(* IEC 61131-3 sources: CodigoPPC/FB Auxiliares, 7 files *)

(* ---- FB_CheckInversores.st ---- *)
// ════════════════════════════════════════════════════════════════════
// FB_CheckInversores — Varredura de presença de inversores no startup
// ════════════════════════════════════════════════════════════════════
//
// Responsabilidade:
//   Percorrer sequencialmente todos os inversores configurados
//   (InvActivePower > 0) em COM1 e COM2, disparar 1 transação
//   Modbus em cada um e verificar ACK. Não valida o valor lido.
//
// Critério de avanço:
//   respondidos / configurados >= GVL_Persis.InvCheckThreshold → xDone=TRUE
//   abaixo do limiar ou timeout global                         → xFailed=TRUE
//
// Contrato com FB_Startup:
//   • xEnable := TRUE  para iniciar/continuar a varredura
//   • xEnable := FALSE reseta o FB (pronto para nova execução)
//   • Lê resultado via xDone / xFailed a cada ciclo
//   • xFailed=TRUE: ler uRespondedTotal e uConfiguredTotal para log
//
// Restrições:
//   • 1 transação Modbus por ciclo de scan (sequencial, determinístico)
//   • Não escreve em GVL_ALARM_MANAGER — responsabilidade do FB_Startup
//   • Tempo máximo: TimeInvTimeout (default 60s para até 30 inversores)
// ════════════════════════════════════════════════════════════════════
FUNCTION_BLOCK FB_CheckInversores

VAR_INPUT
    xEnable         : BOOL;             // TRUE = executar; FALSE = reset
    tTxTimeout      : TIME := T#500MS;  // timeout por transação individual
    tGlobalTimeout  : TIME := T#60S;    // timeout para varredura completa
END_VAR

VAR_OUTPUT
    xDone           : BOOL;             // varredura concluída e acima do limiar
    xFailed         : BOOL;             // abaixo do limiar ou timeout global
    uRespondedTotal : UINT;             // total de inversores que responderam
    uConfiguredTotal: UINT;             // total de inversores configurados
    uLastFailIdx    : UINT;             // índice do último inversor que não respondeu
    uLastFailCOM    : UINT;             // canal do último inversor que não respondeu (1 ou 2)
END_VAR

VAR
    fbTx            : FB_ModBus;        // instância única reutilizada ciclo a ciclo
    uCheckIdx       : UINT := 1;        // índice atual (1..15 dentro do canal)
    uCheckCOM       : UINT := 1;        // canal atual: 1=COM1, 2=COM2, 3=avaliação final
    uRespondedCOM1  : UINT := 0;
    uRespondedCOM2  : UINT := 0;
    bInitDone       : BOOL := FALSE;    // guarda de inicialização
    TonGlobal       : TON;
    // ── Startup: verificação de presença de inversores ────────────
    // Fração mínima de inversores que devem responder para avançar o startup.
    // 1.0 = todos devem responder (padrão conservador)
    // 0.8 = pelo menos 80% devem responder
    CheckThreshold  : REAL := 1.0;
END_VAR

    // ── Reset quando desabilitado ─────────────────────────────────────
    IF NOT xEnable THEN
        xDone            := FALSE;
        xFailed          := FALSE;
        uRespondedCOM1   := 0;
        uRespondedCOM2   := 0;
        uRespondedTotal  := 0;
        uConfiguredTotal := 0;
        uLastFailIdx     := 0;
        uLastFailCOM     := 0;
        uCheckIdx        := 1;
        uCheckCOM        := 1;
        bInitDone        := FALSE;
        TonGlobal(IN := FALSE);
        RETURN;
    END_IF

    // ── Se já terminou, mantém resultado sem re-executar ─────────────
    IF xDone OR xFailed THEN
        RETURN;
    END_IF

    // ── Inicialização na primeira entrada ────────────────────────────
    IF NOT bInitDone THEN
        uConfiguredTotal := GVL_Main.NInversoresCOM01 + GVL_Main.NInversoresCOM02;
        bInitDone        := TRUE;

        // COM2 vazio é permitido — varredura só em COM1
        // uCheckCOM já = 1, sem ação adicional
    END_IF

    // ── Timeout global ────────────────────────────────────────────────
    TonGlobal(IN := TRUE, PT := tGlobalTimeout);
    IF TonGlobal.Q THEN
        TonGlobal(IN := FALSE);
        uRespondedTotal := uRespondedCOM1 + uRespondedCOM2;
        xFailed := TRUE;
        RETURN;
    END_IF

    // ── Varredura COM1 ────────────────────────────────────────────────
    IF uCheckCOM = 1 THEN

        IF uCheckIdx <= GVL_Main.NInversoresCOM01 THEN
            fbTx(
                tTimeout := tTxTimeout,
                trigInv  := GVL_Main.trigInvCOM100[uCheckIdx, 0],
                pSlave   := GVL_Main.pInversores100[uCheckIdx]^
            );

            CASE fbTx.result OF
                E_ModbusResult.DONE:
                    uRespondedCOM1 := uRespondedCOM1 + 1;
                    uCheckIdx      := uCheckIdx + 1;

                E_ModbusResult.ERRO,
                E_ModbusResult.TIMEOUT:
                    uLastFailIdx := uCheckIdx;
                    uLastFailCOM := 1;
                    uCheckIdx    := uCheckIdx + 1;

                // BUSY: aguarda sem avançar
            END_CASE

        ELSE
            // COM1 concluída
            uCheckIdx := 1;
            uCheckCOM := 2;  // avança para COM2 (mesmo que vazia — avaliação em uCheckCOM=3)
        END_IF

    // ── Varredura COM2 ────────────────────────────────────────────────
    ELSIF uCheckCOM = 2 THEN

        IF GVL_Main.NInversoresCOM02 = 0 THEN
            // Canal vazio — pula direto para avaliação
            uCheckCOM := 3;

        ELSIF uCheckIdx <= GVL_Main.NInversoresCOM02 THEN
            fbTx(
                tTimeout := tTxTimeout,
                trigInv  := GVL_Main.trigInvCOM200[uCheckIdx, 0],
                pSlave   := GVL_Main.pInversores200[uCheckIdx]^
            );

            CASE fbTx.result OF
                E_ModbusResult.DONE:
                    uRespondedCOM2 := uRespondedCOM2 + 1;
                    uCheckIdx      := uCheckIdx + 1;

                E_ModbusResult.ERRO,
                E_ModbusResult.TIMEOUT:
                    uLastFailIdx := uCheckIdx;
                    uLastFailCOM := 2;
                    uCheckIdx    := uCheckIdx + 1;

                // BUSY: aguarda sem avançar
            END_CASE

        ELSE
            // COM2 concluída
            uCheckCOM := 3;
        END_IF

    // ── Avaliação final ───────────────────────────────────────────────
    ELSIF uCheckCOM = 3 THEN

        TonGlobal(IN := FALSE);
        uRespondedTotal := uRespondedCOM1 + uRespondedCOM2;

        IF uConfiguredTotal = 0 THEN
            // Proteção defensiva — não deveria chegar aqui (stInit já bloqueia)
            xFailed := TRUE;
            RETURN;
        END_IF

        IF (TO_REAL(uRespondedTotal) / TO_REAL(uConfiguredTotal)) >= CheckThreshold THEN
            xDone := TRUE;
        ELSE
            xFailed := TRUE;
        END_IF

    END_IF

END_FUNCTION_BLOCK

(* ---- FB_ModBus.st ---- *)
FUNCTION_BLOCK FB_ModBus

VAR_INPUT
    tTimeout    : TIME;
END_VAR

VAR_IN_OUT
    trigInv     : BOOL;                    // ex.: Global.trigInvCOM100[i]
    pSlave      : ModbusSlaveComPort;      // ex.: Global.pInversores100[i]^
END_VAR

VAR_OUTPUT
    result      : E_ModbusResult;
END_VAR

VAR
    state       : (TRIG, WAIT_BUSY_ON, WAIT_DONE) := TRIG;
    tonTimer    : TON;
END_VAR

    // ============================================================
    // Máquina de estados de escrita em inversores
    // ============================================================

    // estado default por ciclo
    result := E_ModbusResult.BUSY;

    // timeout só enquanto espera finalização real
    tonTimer(IN := (state = WAIT_DONE), PT := tTimeout);

    CASE state OF

        TRIG:
            trigInv := TRUE;
            state := WAIT_BUSY_ON;

       WAIT_BUSY_ON:
            trigInv := FALSE;            // desce trigger (garante borda)
            IF pSlave.xBusy THEN         // transação realmente iniciou
                state := WAIT_DONE;
            END_IF

        WAIT_DONE:
        	IF pSlave.xDone THEN
                trigInv := FALSE;
                state := TRIG;
                result := E_ModbusResult.DONE;

          	ELSIF pSlave.xError THEN
                state := TRIG;
    			trigInv := FALSE;
                result := E_ModbusResult.ERRO;
    			FC_LogEvent(
    				eCode:=TO_UINT(pSlave.byModbusError) + 16#4A00,
    				bRaised:=TRUE,
    				rParam1:=0.0,
    				rParam2:=0.0,
    				uMachState := GVL_Main.MachineState
    				);

          	ELSIF tonTimer.Q THEN
                state := TRIG;
                trigInv := FALSE;
                result := E_ModbusResult.TIMEOUT;
            END_IF
    END_CASE
END_FUNCTION_BLOCK

(* ---- FB_SetRTC.st ---- *)
(*
================================================================================
  FB_SetRTC — Correção de Data/Hora do RTC via IHM
================================================================================
  Propósito:
    Permite que o operador corrija o relógio do CLP (WAGO CC100) diretamente
    pela IHM, sem necessidade de acesso ao Codesys IDE.

  Problema resolvido:
    O CC100 não possui bateria de RTC confiável. Após queda de energia, o
    relógio retorna para 1970-01-01 00:00:00. Isso corrompe o agendamento
    (FB_Scheduler), o log de eventos e qualquer registro com timestamp.

  Comportamento:
    1. O operador preenche os campos de data/hora na IHM e aciona bSet=TRUE.
    2. O FB valida todos os campos antes de qualquer escrita.
    3. Se válido: chama SysTimeRtcSet(), registra evento INFO no log.
    4. Se inválido: recusa a operação, registra WARNING com o campo problemático.
    5. bSet é um pulso de borda de subida — consumido internamente (auto-reset).
    6. bBusy permanece TRUE por 1 ciclo após a operação para sinalizar atividade.
    7. bSuccess e bError são mantidos por FEEDBACK_HOLD_CYCLES ciclos.

  Integração:
    - Chamar em TaskIHM (não na task de controle — operação pontual, não crítica).
    - Expor todas as variáveis VAR_INPUT/OUTPUT na tela de configuração da IHM.
    - A task de controle NÃO precisa ser modificada.

  Notas de segurança:
    - O FB NÃO impede a máquina de estados de operar durante a atualização.
    - SysTimeRtcSet() é atômico no WAGO CC100 / Codesys V3.5.
    - Ano mínimo: 2020 (evita aceitar 1970 de RTC sem bateria).
    - Ano máximo: 2099 (limite de UDINT epoch seguro).
    - O FB não aceita segundos bissextos (segundo 60) — simplificação segura.

  Dependências:
    - SysTimeRtc.library (SysTimeRtcSet, SysTimeRtcGet, SysTimeRtcConvertDateToUTC)
    - FC_LogEvent, E_EventCode, GVL_Main
    - Codesys V3.5 SP21 / IEC 61131-3 Structured Text

  Revisão: 2026-03
================================================================================
*)
FUNCTION_BLOCK FB_SetRTC

VAR_INPUT
    // ── Comando ───────────────────────────────────────────────────────────────
    bSet        : BOOL;     // Pulso de subida = aplica nova data/hora
                            // IHM deve manter TRUE por ≥ 1 ciclo, depois FALSE

    // ── Data/Hora desejada (preenchida pelo operador na IHM) ──────────────────
    nYear       : UINT;     // Ano   [2020 .. 2099]
    nMonth      : UINT;     // Mês   [1 .. 12]
    nDay        : UINT;     // Dia   [1 .. 31] (validação completa por mês)
    nHour       : UINT;     // Hora  [0 .. 23]
    nMinute     : UINT;     // Min   [0 .. 59]
    nSecond     : UINT;     // Seg   [0 .. 59]
END_VAR

VAR_OUTPUT
    // ── Feedback para a IHM ───────────────────────────────────────────────────
    bBusy           : BOOL;     // TRUE durante o ciclo de execução
    bSuccess        : BOOL;     // TRUE por FEEDBACK_HOLD_CYCLES após sucesso
    bError          : BOOL;     // TRUE por FEEDBACK_HOLD_CYCLES após falha
    nErrorCode      : UINT;     // Código do erro (ver constantes abaixo):
                                //   0 = sem erro
                                //   1 = Ano inválido
                                //   2 = Mês inválido
                                //   3 = Dia inválido para o mês/ano
                                //   4 = Hora inválida
                                //   5 = Minuto inválido
                                //   6 = Segundo inválido
                                //   7 = SysTimeRtcSet() falhou (erro de hardware)
    sStatusMsg      : STRING(40); // Mensagem legível para display na IHM
END_VAR

VAR
    // ── Detecção de borda de subida em bSet ───────────────────────────────────
    rTrigSet        : R_TRIG;

    // ── Variáveis para cálculo de epoch e chamada de SysTimeRtcSet ──────────
    // SysTimeRtcSet(ulTimestamp: DWORD): RTS_IEC_RESULT
    // Recebe segundos desde 1970-01-01 00:00:00 UTC (epoch Unix).
    ulTimestamp     : UDINT;            // Epoch calculado a partir dos campos da IHM
    rtcResult       : RTS_IEC_RESULT;

    // ── Variáveis auxiliares para cálculo de epoch ────────────────────────────
    nY              : UDINT;            // Ano de trabalho (loop)
    nDays           : UDINT;            // Acumulador de dias desde 1970

    // ── Contador de ciclos para manter feedback visível na IHM ───────────────
    nFeedbackTimer  : UINT;

    // ── Dias por mês (índice 1..12) — fevereiro = 28; bissexto tratado em código
    aDaysInMonth    : ARRAY[1..12] OF UINT
                    := [31, 28, 31, 30, 31, 30, 31, 31, 30, 31, 30, 31];

    // ── Constante: quantos ciclos manter bSuccess/bError visíveis ─────────────
    // Com CYCLE_TIME_MS = 1000 ms → 5 ciclos = 5 segundos de feedback
    FEEDBACK_HOLD_CYCLES : UINT := 5;
END_VAR

    // ════════════════════════════════════════════════════════════════════════════
    // 1. DETECÇÃO DE BORDA — garante execução única por pulso do operador
    // ════════════════════════════════════════════════════════════════════════════
    rTrigSet(CLK := bSet);

    // ════════════════════════════════════════════════════════════════════════════
    // 2. TEMPORIZADOR DE FEEDBACK — mantém bSuccess/bError visíveis por N ciclos
    // ════════════════════════════════════════════════════════════════════════════
    IF nFeedbackTimer > 0 THEN
        nFeedbackTimer := nFeedbackTimer - 1;
        IF nFeedbackTimer = 0 THEN
            bSuccess := FALSE;
            bError   := FALSE;
            nErrorCode := 0;
            sStatusMsg := 'Aguardando comando...';
        END_IF
    END_IF

    // ════════════════════════════════════════════════════════════════════════════
    // 3. EXECUÇÃO — apenas na borda de subida de bSet
    // ════════════════════════════════════════════════════════════════════════════
    IF NOT rTrigSet.Q THEN
        RETURN;
    END_IF

    // ── Sinaliza ocupado neste ciclo ─────────────────────────────────────────
    bBusy    := TRUE;
    bSuccess := FALSE;
    bError   := FALSE;
    nErrorCode := 0;

    // ════════════════════════════════════════════════════════════════════════════
    // 4. VALIDAÇÃO DOS CAMPOS
    // ════════════════════════════════════════════════════════════════════════════

    // 4.1 Ano — aceita apenas datas a partir de 2020 para rejeitar RTC sem bateria
    IF nYear < 2020 OR nYear > 2099 THEN
        nErrorCode := 1;
        bError     := TRUE;
        sStatusMsg := 'ERRO: Ano invalido (2020-2099)';
        nFeedbackTimer := FEEDBACK_HOLD_CYCLES;
        bBusy := FALSE;
        FC_LogEvent(
            eCode      := E_EventCode.WARN_RTC_SET_INVALID_INPUT,
            bRaised    := TRUE,
            rParam1    := TO_REAL(nYear),
            rParam2    := 1.0,
            uMachState := GVL_Main.MachineState
        );
        RETURN;
    END_IF

    // 4.2 Mês
    IF nMonth < 1 OR nMonth > 12 THEN
        nErrorCode := 2;
        bError     := TRUE;
        sStatusMsg := 'ERRO: Mes invalido (1-12)';
        nFeedbackTimer := FEEDBACK_HOLD_CYCLES;
        bBusy := FALSE;
        FC_LogEvent(
            eCode      := E_EventCode.WARN_RTC_SET_INVALID_INPUT,
            bRaised    := TRUE,
            rParam1    := TO_REAL(nMonth),
            rParam2    := 2.0,
            uMachState := GVL_Main.MachineState
        );
        RETURN;
    END_IF

    // 4.3 Dia — considera ano bissexto para fevereiro
    // Ano bissexto: divisível por 4, exceto centenários não divisíveis por 400
    IF nMonth = 2 THEN
        IF ((nYear MOD 4 = 0) AND (nYear MOD 100 <> 0)) OR (nYear MOD 400 = 0) THEN
            aDaysInMonth[2] := 29;  // Fevereiro tem 29 dias neste ano
        ELSE
            aDaysInMonth[2] := 28;
        END_IF
    END_IF

    IF nDay < 1 OR nDay > aDaysInMonth[nMonth] THEN
        nErrorCode := 3;
        bError     := TRUE;
        sStatusMsg := 'ERRO: Dia invalido para o mes/ano';
        nFeedbackTimer := FEEDBACK_HOLD_CYCLES;
        bBusy := FALSE;
        FC_LogEvent(
            eCode      := E_EventCode.WARN_RTC_SET_INVALID_INPUT,
            bRaised    := TRUE,
            rParam1    := TO_REAL(nDay),
            rParam2    := 3.0,
            uMachState := GVL_Main.MachineState
        );
        RETURN;
    END_IF

    // 4.4 Hora
    IF nHour > 23 THEN
        nErrorCode := 4;
        bError     := TRUE;
        sStatusMsg := 'ERRO: Hora invalida (0-23)';
        nFeedbackTimer := FEEDBACK_HOLD_CYCLES;
        bBusy := FALSE;
        FC_LogEvent(
            eCode      := E_EventCode.WARN_RTC_SET_INVALID_INPUT,
            bRaised    := TRUE,
            rParam1    := TO_REAL(nHour),
            rParam2    := 4.0,
            uMachState := GVL_Main.MachineState
        );
        RETURN;
    END_IF

    // 4.5 Minuto
    IF nMinute > 59 THEN
        nErrorCode := 5;
        bError     := TRUE;
        sStatusMsg := 'ERRO: Minuto invalido (0-59)';
        nFeedbackTimer := FEEDBACK_HOLD_CYCLES;
        bBusy := FALSE;
        FC_LogEvent(
            eCode      := E_EventCode.WARN_RTC_SET_INVALID_INPUT,
            bRaised    := TRUE,
            rParam1    := TO_REAL(nMinute),
            rParam2    := 5.0,
            uMachState := GVL_Main.MachineState
        );
        RETURN;
    END_IF

    // 4.6 Segundo — rejeita segundo 60 (bissexto): simplificação segura para CLP
    IF nSecond > 59 THEN
        nErrorCode := 6;
        bError     := TRUE;
        sStatusMsg := 'ERRO: Segundo invalido (0-59)';
        nFeedbackTimer := FEEDBACK_HOLD_CYCLES;
        bBusy := FALSE;
        FC_LogEvent(
            eCode      := E_EventCode.WARN_RTC_SET_INVALID_INPUT,
            bRaised    := TRUE,
            rParam1    := TO_REAL(nSecond),
            rParam2    := 6.0,
            uMachState := GVL_Main.MachineState
        );
        RETURN;
    END_IF

    // ════════════════════════════════════════════════════════════════════════════
    // 5. CONVERTE DATA/HORA PARA EPOCH UNIX E CHAMA SysTimeRtcSet()
    // ════════════════════════════════════════════════════════════════════════════
    // A data/hora informada pelo operador na IHM é UTC (sem offset de fuso).
    // Justificativa: o sistema já trata fuso internamente no FB_Scheduler.
    //
    // Algoritmo: conta dias desde 1970-01-01, aplica horas/min/seg.
    // Validado para o intervalo 2020..2099 — sem risco de overflow em UDINT.
    //
    // SysTimeRtcSet(ulTimestamp: DWORD): RTS_IEC_RESULT
    // Fonte confirmada: SysTimeRtc.library Codesys V3.5 — assinatura real do target.

    // 5.1 Acumula dias dos anos completos desde 1970 até (nYear - 1)
    nDays := 0;
    FOR nY := 1970 TO UINT_TO_UDINT(nYear) - 1 DO
        IF ((nY MOD 4 = 0) AND (nY MOD 100 <> 0)) OR (nY MOD 400 = 0) THEN
            nDays := nDays + 366;   // Ano bissexto
        ELSE
            nDays := nDays + 365;
        END_IF
    END_FOR

    // 5.2 Acumula dias dos meses completos no ano corrente (1..nMonth-1)
    // aDaysInMonth[2] já foi corrigido para 29 se bissexto (seção 4.3)
    IF nMonth > 1  THEN nDays := nDays + UINT_TO_UDINT(aDaysInMonth[1]);  END_IF
    IF nMonth > 2  THEN nDays := nDays + UINT_TO_UDINT(aDaysInMonth[2]);  END_IF
    IF nMonth > 3  THEN nDays := nDays + UINT_TO_UDINT(aDaysInMonth[3]);  END_IF
    IF nMonth > 4  THEN nDays := nDays + UINT_TO_UDINT(aDaysInMonth[4]);  END_IF
    IF nMonth > 5  THEN nDays := nDays + UINT_TO_UDINT(aDaysInMonth[5]);  END_IF
    IF nMonth > 6  THEN nDays := nDays + UINT_TO_UDINT(aDaysInMonth[6]);  END_IF
    IF nMonth > 7  THEN nDays := nDays + UINT_TO_UDINT(aDaysInMonth[7]);  END_IF
    IF nMonth > 8  THEN nDays := nDays + UINT_TO_UDINT(aDaysInMonth[8]);  END_IF
    IF nMonth > 9  THEN nDays := nDays + UINT_TO_UDINT(aDaysInMonth[9]);  END_IF
    IF nMonth > 10 THEN nDays := nDays + UINT_TO_UDINT(aDaysInMonth[10]); END_IF
    IF nMonth > 11 THEN nDays := nDays + UINT_TO_UDINT(aDaysInMonth[11]); END_IF
    // Mês 12 não tem mês seguinte — não precisa de entrada aqui

    // 5.3 Adiciona os dias completos do mês atual (nDay - 1)
    nDays := nDays + UINT_TO_UDINT(nDay) - 1;

    // 5.4 Converte dias + horas + min + seg para epoch em segundos
    ulTimestamp := (nDays * 86400)
                 + (UINT_TO_UDINT(nHour)   * 3600)
                 + (UINT_TO_UDINT(nMinute) * 60)
                 +  UINT_TO_UDINT(nSecond);

    // 5.5 Chama SysTimeRtcSet com o epoch calculado
    rtcResult := SysTimeRtcSet(ulTimestamp := UDINT_TO_DWORD(ulTimestamp));

    // ════════════════════════════════════════════════════════════════════════════
    // 6. VERIFICA RESULTADO DE SysTimeRtcSet()
    // ════════════════════════════════════════════════════════════════════════════
    IF rtcResult <> 0 THEN
        nErrorCode := 7;
        bError     := TRUE;
        sStatusMsg := 'ERRO: Falha no hardware RTC';
        nFeedbackTimer := FEEDBACK_HOLD_CYCLES;
        bBusy := FALSE;
        FC_LogEvent(
            eCode      := E_EventCode.WARN_RTC_SET_HW_FAIL,
            bRaised    := TRUE,
            rParam1    := UINT_TO_REAL(TO_UINT(rtcResult)),
            rParam2    := 0.0,
            uMachState := GVL_Main.MachineState
        );
        RETURN;
    END_IF

    // ════════════════════════════════════════════════════════════════════════════
    // 7. SUCESSO — atualiza GVL_Main.timestampUTC imediatamente
    //    (evita 1 ciclo com timestamp antigo no FB_Scheduler)
    // ════════════════════════════════════════════════════════════════════════════
    GVL_Main.timestampUTC := TO_UDINT(SysTimeRtcGet(GVL_Main.Result));

    bSuccess       := TRUE;
    sStatusMsg     := 'RTC atualizado com sucesso';
    nFeedbackTimer := FEEDBACK_HOLD_CYCLES;
    bBusy          := FALSE;

    FC_LogEvent(
        eCode      := E_EventCode.INFO_RTC_SET_OK,
        bRaised    := TRUE,
        rParam1    := UINT_TO_REAL(nYear) * 10000.0
                   + UINT_TO_REAL(nMonth) * 100.0
                   + UINT_TO_REAL(nDay),       // Ex: 20260306 → codifica AAAAMMDD
        rParam2    := UINT_TO_REAL(nHour) * 10000.0
                   + UINT_TO_REAL(nMinute) * 100.0
                   + UINT_TO_REAL(nSecond),    // Ex: 143015 → codifica HHMMSS
        uMachState := GVL_Main.MachineState
    );
END_FUNCTION_BLOCK

(* ---- FB_Startup.st ---- *)
(* ════════════════════════════════════════════════════════════════════
   FB_Startup — Sequência de inicialização do PPC-GD
   ════════════════════════════════════════════════════════════════════
   Sequência de estados:
     stInit             → cálculos iniciais: RTC, ciclo, ponteiros,
                          contagem de inversores, potência instalada
     stCheck_COM        → aguarda driver Modbus RTU atingir RUNNING
     stCheck_Medidor    → confirma ACK Modbus do medidor
     stCheck_Inversores → varredura de presença nos inversores
     stWait_K1          → fecha K1_out; aguarda K1_in com debounce
     stWait_K2          → aguarda K2_in com debounce
     stDone             → startup concluído → MainProgram vai para IDLE
     stError            → falha de startup  → MainProgram vai para STOP

   Notas:
     - K1_in e K2_in devem ser contatos auxiliares dos disjuntores.
       Se não forem usados contatos auxiliares, conectar a 24V.
     - Este FB controla K1_out e os LEDs. K2_out é controlado pelo
       MainProgram (estado STOP).
     - TONs devem ser chamados todo ciclo para acumular tempo
       corretamente — nunca instanciar dentro de IF.
   ════════════════════════════════════════════════════════════════════ *)

FUNCTION_BLOCK FB_Startup

VAR_OUTPUT
    stState             : E_StartupStatus := E_StartupStatus.stInit;
END_VAR

VAR
    // ── Entradas digitais (lidas no início de cada ciclo) ─────────
    auxK1_in            : BOOL;                     // espelho de GVL_Main.K1_in
    auxK2_in            : BOOL;                     // espelho de GVL_Main.K2_in

    // ── Saídas físicas (calculadas no corpo, aplicadas no final) ──
    cmdK01              : BOOL := FALSE;            // K1_out
    auxRed              : BOOL := FALSE;            // LedRedOut
    auxYellow           : BOOL := FALSE;            // LedYellowOut
    auxGreen            : BOOL := FALSE;            // LedGreenOut

    // ── Variável de loop (stInit) ─────────────────────────────────
    indice              : UINT;

    // ── stCheck_COM: aguarda driver Modbus RTU ────────────────────
    eDeviceState01      : DED.DEVICE_STATE;         // estado retornado pelo Master_01
    xDiagInfo01         : BOOL;                     // xDiagnosisInfoAvailable do Master_01
    eError01            : DED.ERROR;                // código de erro do Master_01
    xMaster01IsReady    : BOOL;                     // TRUE quando Master_01 = RUNNING

    eDeviceState02      : DED.DEVICE_STATE;         // estado retornado pelo Master_02
    xDiagInfo02         : BOOL;                     // xDiagnosisInfoAvailable do Master_02
    eError02            : DED.ERROR;                // código de erro do Master_02
    xMaster02IsReady    : BOOL;                     // TRUE quando Master_02 = RUNNING

    TonComTimeout       : TON;                      // timeout de espera pelo driver
    TimeComTimeout      : TIME := T#10S;            // 10s: conservador para boot do driver RTU
    bComLogSent         : BOOL := FALSE;            // evita log repetido de INFO_SERIAL_COM_OK

    // ── stCheck_Medidor: confirma ACK Modbus do medidor ───────────
    fbDiagMedidor       : FB_ModBus;                // transação de diagnóstico do medidor
    TonMedTimeout       : TON;                      // timeout global da verificação
    TimeMedTimeout      : TIME := T#10S;            // 10s: margem para medidor lento

    // ── stCheck_Inversores: varredura de presença ─────────────────
    fbCheckInv          : FB_CheckInversores;       // varredura sequencial por ACK Modbus

    // ── stWait_K1: debounce e timeout de K1 ──────────────────────
    debouncedK1         : BOOL := FALSE;            // TRUE quando K1_in estável por TimeDebounceK1
    TonDebounceK1       : TON;                      // acumula tempo de estabilidade de K1_in
    TimeDebounceK1      : TIME := T#500MS;          // tempo mínimo de estabilidade para K1
    TonK1Timeout        : TON;                      // timeout máximo aguardando K1 fechar
    TimeK1Timeout       : TIME := T#5S;             // tempo máximo para K1 responder

    // ── stWait_K2: debounce e timeout de K2 ──────────────────────
    debouncedK2         : BOOL := FALSE;            // TRUE quando K2_in estável por TimeDebounceK2
    TonDebounceK2       : TON;                      // acumula tempo de estabilidade de K2_in
    TimeDebounceK2      : TIME := T#500MS;          // tempo mínimo de estabilidade para K2
    TonK2Timeout        : TON;                      // timeout máximo aguardando K2 fechar
    TimeK2Timeout       : TIME := T#5S;             // tempo máximo para K2 responder

END_VAR

    // INICIA AQUI

    auxK1_in := GVL_Main.K1_in;
    auxK2_in := GVL_Main.K2_in;

    CASE stState OF 																				// Máquina de estados

    	// ────────────────────────────────────────────────────────────
    	// ────────────────────────────────────────────────────────────
    	E_StartupStatus.stInit:																		// Inicialização única

    		cmdK01 			:= FALSE;
    		auxRed  		:= FALSE;
    		auxYellow 		:= FALSE;
    		auxGreen  		:= FALSE;
    		debouncedK1 	:= FALSE;
    		debouncedK2 	:= FALSE;

    		// Testa leitura do relógio do sistema na inicialização
    		GVL_Main.timestampUTC := TO_UDINT(SysTimeRtcGet(GVL_Main.Result)); 							// UDINT#1528268918
    		GVL_Alarm.CRIT_RTC_FAIL:=(GVL_Main.Result <> eResultCode.OK);                        // Em caso de erro de leitura do relógio, vai para STOP
    		IF GVL_Alarm.CRIT_RTC_FAIL THEN
    			GVL_Main.LedRedOut:=TRUE;																// sinalizar que houve erro para ler o relógio
    			FC_LogEvent(
    				eCode      := E_EventCode.CRIT_RTC_FAILED,
    				bRaised    := TRUE,
    				rParam1    := 0.0,
    				rParam2    := 0.0,
    				uMachState := GVL_Main.MachineState
    			);
    			stState := E_StartupStatus.stError;
    			RETURN;
    		END_IF

    		// -----------------------------------------------------------------------------------------
    		// PREPARAÇÃO DO TEMPO DE CICLO - feito na inicialização

    		// Converte TIME (ex: T#500ms) para REAL (0.5 segundos) para uso nos PIDs
    		GVL_Main.ControlCycle := UDINT_TO_REAL(GVL_Main.CYCLE_TIME_MS)/1000;  				// converte para segundos
    		GVL_Main.CYCLE_TIME_TOLERANCE:=TO_UDINT(TO_REAL(GVL_Main.CYCLE_TIME_MS)*1.2);

    		// -----------------------------------------------------------------------------------------
    		// Porta de comunicação COM1
    		GVL_Main.pMedidor100   		:= ADR(Medidor100);
    		GVL_Main.pInversores100[1]  := ADR(Inversor101);
    		GVL_Main.pInversores100[2]  := ADR(Inversor102);
    		GVL_Main.pInversores100[3]	:= ADR(Inversor103);
    		GVL_Main.pInversores100[4] 	:= ADR(Inversor104);
    		GVL_Main.pInversores100[5]	:= ADR(Inversor105);
    		GVL_Main.pInversores100[6] 	:= ADR(Inversor106);
    		GVL_Main.pInversores100[7] 	:= ADR(Inversor107);
    		GVL_Main.pInversores100[8] 	:= ADR(Inversor108);
    		GVL_Main.pInversores100[9] 	:= ADR(Inversor109);
    		GVL_Main.pInversores100[10]	:= ADR(Inversor110);
    		GVL_Main.pInversores100[11]	:= ADR(Inversor111);
    		GVL_Main.pInversores100[12] := ADR(Inversor112);
    		GVL_Main.pInversores100[13] := ADR(Inversor113);
    		GVL_Main.pInversores100[14] := ADR(Inversor114);
    		GVL_Main.pInversores100[15] := ADR(Inversor115);

    		// Porta de comunicação COM2
    		GVL_Main.pMedidor200   	  	:= ADR(Medidor200);
    		GVL_Main.pInversores200[1]  := ADR(Inversor201);
    		GVL_Main.pInversores200[2]  := ADR(Inversor202);
    		GVL_Main.pInversores200[3]  := ADR(Inversor203);
    		GVL_Main.pInversores200[4]  := ADR(Inversor204);
    		GVL_Main.pInversores200[5] 	:= ADR(Inversor205);
    		GVL_Main.pInversores200[6]  := ADR(Inversor206);
    		GVL_Main.pInversores200[7]  := ADR(Inversor207);
    		GVL_Main.pInversores200[8]  := ADR(Inversor208);
    		GVL_Main.pInversores200[9]  := ADR(Inversor209);
    		GVL_Main.pInversores200[10] := ADR(Inversor210);
    		GVL_Main.pInversores200[11] := ADR(Inversor211);
    		GVL_Main.pInversores200[12] := ADR(Inversor212);
    		GVL_Main.pInversores200[13] := ADR(Inversor213);
    		GVL_Main.pInversores200[14] := ADR(Inversor214);
    		GVL_Main.pInversores200[15] := ADR(Inversor215);

    		// -----------------------------------------------------------------------------------------
    		// CONTAGEM AUTOMÁTICA DE INVERSORES (sequencial por potência)

    		// COM1: índices 1..15
    		GVL_Main.NInversoresCOM01 := 0;
    		FOR indice := 1 TO 15 DO
    			IF GVL_Pers.InvActivePower[indice] > 0.0 THEN
    				GVL_Main.NInversoresCOM01 := indice;   // mantém maior índice válido
    			ELSE
    				EXIT;  // encontrou buraco -> encerra contagem
    			END_IF
    		END_FOR

    		// COM2: índices 16..30
    		GVL_Main.NInversoresCOM02 := 0;
    		FOR indice := 16 TO 30 DO
    			IF GVL_Pers.InvActivePower[indice] > 0.0 THEN
    				GVL_Main.NInversoresCOM02 := indice - 15;   // converte para faixa 1..15
    			ELSE
    				EXIT;  // encontrou buraco -> encerra contagem
    			END_IF
    		END_FOR

    		GVL_Main.MAX_CH1_MODBUS_ERROS		:= GVL_Main.NInversoresCOM01 / 2;					// permite < 50% da quantidade de inversores sem ir para FAIL
    		GVL_Main.MAX_CH1_MODBUS_TIMEOUTS	:= GVL_Main.NInversoresCOM01 / 2;					// permite < 50% da quantidade de inversores sem ir para FAIL
    		GVL_Main.MAX_CH2_MODBUS_ERROS		:= GVL_Main.NInversoresCOM02 / 2;					// permite < 50% da quantidade de inversores sem ir para FAIL
    		GVL_Main.MAX_CH2_MODBUS_TIMEOUTS	:= GVL_Main.NInversoresCOM02 / 2;					// permite < 50% da quantidade de inversores sem ir para FAIL

    		// -----------------------------------------------------------------------------------------
    		// CÁLCULO DA POTÊNCIA INSTALADA TOTAL (Ativa e Aparente)  - feito na inicialização

    		// Soma a capacidade nominal de todos os inversores configurados.
    		// Isso permite mudar a planta dinamicamente sem recompilar.

    		GVL_Main.InstalledPower := 0.0;
    		GVL_Main.InstalledSmax  := 0.0;

    		FOR indice := 1 TO GVL_Main.NMAXINVERSORES DO
    			// Soma Potência Ativa Máxima (kW)
    			GVL_Main.InstalledPower := GVL_Main.InstalledPower + GVL_Pers.InvActivePower[indice];
    			// Soma Potência Aparente Máxima (kVA)
    			GVL_Main.InstalledSmax := GVL_Main.InstalledSmax + GVL_Pers.InvSmaxPower[indice];
    		END_FOR

    		// Se não houver inversores ou potência válida, zera tudo e sai

    		GVL_Alarm.CRIT_INSTALLED_PWR_ZERO:= (GVL_Main.InstalledPower <= 0.0);
    		IF GVL_Alarm.CRIT_INSTALLED_PWR_ZERO THEN
    			GVL_Main.TotalReactivePower := 0.0;
    			GVL_Main.LedRedOut:=TRUE;
    			stState := E_StartupStatus.stError;
    			FC_LogEvent(
    				eCode      := E_EventCode.CRIT_INSTALLED_PWR_ZERO,
    				bRaised    := TRUE,
    				rParam1    := GVL_Main.TotalReactivePower,
    				rParam2    := 0.0,
    				uMachState := GVL_Main.MachineState
    			);
    			stState := E_StartupStatus.stError;
    			RETURN;
    		END_IF

    		GVL_Alarm.CRIT_INSTALLED_SMAX_ZERO:= (GVL_Main.InstalledSmax <= 0.0);
    		IF GVL_Alarm.CRIT_INSTALLED_SMAX_ZERO THEN
    			GVL_Main.TotalReactivePower := 0.0;
    			GVL_Main.LedRedOut:=TRUE;
    			stState := E_StartupStatus.stError;
    			FC_LogEvent(
    				eCode      := E_EventCode.CRIT_INSTALLED_SMAX_ZERO,
    				bRaised    := TRUE,
    				rParam1    := GVL_Main.TotalReactivePower,
    				rParam2    := 0.0,
    				uMachState := GVL_Main.MachineState
    			);
    			stState := E_StartupStatus.stError;
    			RETURN;
    		END_IF

    		// Calcula Q_max_permitido
    	    GVL_Main.Q_max_permitido := GVL_Main.InstalledPower * 0.4256;  						// tan(acos(0.92))

    		// Configura TC_Power_kW se não foi configurado
    		GVL_Alarm.CRIT_TC_POWER_NOT_SET:=(GVL_Pers.TC_Power_kW = 0.0);
    		IF GVL_Alarm.CRIT_TC_POWER_NOT_SET THEN
    			GVL_Pers.TC_Power_kW := GVL_Main.InstalledPower;  							// Aproximação conservadora
    			stState := E_StartupStatus.stError;
    			FC_LogEvent(
    				eCode      := E_EventCode.CRIT_TC_POWER_NOT_SET,
    				bRaised    := TRUE,
    				rParam1    := GVL_Pers.TC_Power_kW,
    				rParam2    := 0.0,
    				uMachState := GVL_Main.MachineState
    			);
    			stState := E_StartupStatus.stError;
    			RETURN;
    		END_IF

    		// zera setpoints por segurança
            FOR indice := 1 TO GVL_Main.NMAXINVERSORES DO
                GVL_Main.P_inv_kW[indice] := 0.0;
                GVL_Main.P_inv_Percent[indice] := 0.0;
                GVL_Main.Q_inv_kvar[indice] := 0.0;
            END_FOR

    		// Muda para próximo estado
    		stState := E_StartupStatus.stCheck_COM;

    	// ────────────────────────────────────────────────────────────
    	// ────────────────────────────────────────────────────────────
    	E_StartupStatus.stCheck_COM:
    	    // ────────────────────────────────────────────────────────────
            // Aguarda o driver Modbus RTU atingir RUNNING em COM1 e COM2.
            // Necessário porque no boot o driver passa por INITIALIZING
            // antes de ficar pronto — verificação única em stInit falharia
            // sistematicamente em power cycles.
            //
            // Permanece aqui até:
            //   a) Ambos RUNNING            → avança para stWait_K1
            //   b) TonComTimeout.Q          → stError (driver não inicializou)
            //
            // LEDs: vermelho piscante não disponível (sem saída PWM).
            // Mantém vermelho sólido durante a espera — estado não operacional.
            // ────────────────────────────────────────────────────────────

            auxRed    := TRUE;
            auxYellow := FALSE;
            auxGreen  := FALSE;
            cmdK01    := FALSE;    // K1 permanece aberto durante verificação

            TonComTimeout(IN := TRUE, PT := TimeComTimeout);

            eDeviceState01 := Master_01.GetDeviceState(
                xDiagnosisInfoAvailable => xDiagInfo01,
                eError                  => eError01
            );
            eDeviceState02 := Master_02.GetDeviceState(
                xDiagnosisInfoAvailable => xDiagInfo02,
                eError                  => eError02
            );
            xMaster01IsReady := (eDeviceState01 = DED.DEVICE_STATE.RUNNING);
            xMaster02IsReady := (eDeviceState02 = DED.DEVICE_STATE.RUNNING);

            IF xMaster01IsReady AND xMaster02IsReady THEN
                // Sucesso: driver pronto em ambas as COMs
                TonComTimeout(IN := FALSE);
                GVL_Alarm.CRIT_SERIAL_INIT_FAIL := FALSE;
                IF NOT bComLogSent THEN
                    FC_LogEvent(
                        eCode      := E_EventCode.INFO_SERIAL_COM_OK,
                        bRaised    := TRUE,
                        rParam1    := 0.0,
                        rParam2    := 0.0,
                        uMachState := GVL_Main.MachineState
                    );
                    bComLogSent := TRUE;
                END_IF
                stState := E_StartupStatus.stWait_K1;

            ELSIF TonComTimeout.Q THEN
                // Falha: driver não atingiu RUNNING dentro do tempo limite
                TonComTimeout(IN := FALSE);
                GVL_Alarm.CRIT_SERIAL_INIT_FAIL := TRUE;
                GVL_Main.LedRedOut := TRUE;
                FC_LogEvent(
                    eCode      := E_EventCode.CRIT_SERIAL_INIT_FAILED,
                    bRaised    := TRUE,
                    rParam1    := BOOL_TO_REAL(NOT xMaster01IsReady),  // 1.0 = COM1 falhou
                    rParam2    := BOOL_TO_REAL(NOT xMaster02IsReady),  // 1.0 = COM2 falhou
                    uMachState := GVL_Main.MachineState
                );
                stState := E_StartupStatus.stError;

            // ELSE: driver ainda em INITIALIZING — permanece neste estado,
            //       TonComTimeout acumulando. Sem ação, sem transição.
            END_IF

    		(* Nota sobre `rParam1`/`rParam2`:**
    		passar `BOOL_TO_REAL(NOT xMaster01IsReady)` codifica qual COM falhou diretamente no evento
    		 — `rParam1=1.0` significa COM1 não subiu, `rParam2=1.0` significa COM2 não subiu.
    		Isso permite diagnóstico imediato sem precisar de outro evento.
    		*)

    	// ────────────────────────────────────────────────────────────
    	// ────────────────────────────────────────────────────────────
    	E_StartupStatus.stCheck_Medidor:
        // Dispara 1 transação de leitura no medidor (trigger de diagnóstico)
        // Aguarda DONE ou ERRO/TIMEOUT com timeout global
        fbDiagMedidor(
            tTimeout := T#2S,
            trigInv  := GVL_Main.trigMedidor100,
            pSlave   := GVL_Main.pMedidor100^
        );
        TonMedTimeout(IN := TRUE, PT :=TimeMedTimeout);

        CASE fbDiagMedidor.result OF
            E_ModbusResult.DONE:
                TonMedTimeout(IN := FALSE);
    			GVL_Alarm.CRIT_MEAS_INIC_ERRO_TIMEOUT := FALSE;
                stState := E_StartupStatus.stCheck_Inversores;

            E_ModbusResult.ERRO,
            E_ModbusResult.TIMEOUT:
                GVL_Alarm.CRIT_MEAS_INIC_ERRO_TIMEOUT := TRUE;
    			FC_LogEvent(
                    eCode      := E_EventCode.CRIT_MEAS_INIC_ERRO_TIMEOUT,
                    bRaised    := TRUE,
                    rParam1    := 0.0,
                    rParam2    := 0.0,
                    uMachState := GVL_Main.MachineState
                );
                stState := E_StartupStatus.stError;
            // BUSY: permanece aguardando
        END_CASE

        IF TonMedTimeout.Q THEN
    		FC_LogEvent(
            	eCode      := E_EventCode.CRIT_MEAS_INIC_FAIL,
                bRaised    := TRUE,
                rParam1    := 0.0,
                rParam2    := 0.0,
                uMachState := GVL_Main.MachineState
                );
            stState := E_StartupStatus.stError;
        END_IF

    	// ────────────────────────────────────────────────────────────
    	// ────────────────────────────────────────────────────────────
    	E_StartupStatus.stCheck_Inversores:
    	// testa comunicação com inversores

            auxRed    := TRUE;
            auxYellow := FALSE;
            auxGreen  := FALSE;
            cmdK01    := FALSE;

            fbCheckInv(xEnable := TRUE);

            IF fbCheckInv.xDone THEN
                fbCheckInv(xEnable := FALSE);  // reset para próxima execução

                IF fbCheckInv.uRespondedTotal < fbCheckInv.uConfiguredTotal THEN
                    // Passou no limiar mas com ausências — warning
                    GVL_Alarm.WARN_INV_CHECK_PARTIAL := TRUE;
                    FC_LogEvent(
                        eCode      := E_EventCode.WARN_INV_CHECK_PARTIAL,
                        bRaised    := TRUE,
                        rParam1    := TO_REAL(fbCheckInv.uRespondedTotal),
                        rParam2    := TO_REAL(fbCheckInv.uConfiguredTotal),
                        uMachState := GVL_Main.MachineState
                    );
                ELSE
                    FC_LogEvent(
                        eCode      := E_EventCode.INFO_INV_CHECK_OK,
                        bRaised    := TRUE,
                        rParam1    := TO_REAL(fbCheckInv.uRespondedTotal),
                        rParam2    := TO_REAL(fbCheckInv.uConfiguredTotal),
                        uMachState := GVL_Main.MachineState
                    );
    				GVL_Alarm.WARN_INV_CHECK_PARTIAL := FALSE;
                	GVL_Alarm.CRIT_INV_CHECK_BELOW_THRESHOLD := FALSE;
                END_IF
                stState := E_StartupStatus.stWait_K1;

            ELSIF fbCheckInv.xFailed THEN
                fbCheckInv(xEnable := FALSE);  // reset

                GVL_Alarm.CRIT_INV_CHECK_BELOW_THRESHOLD := TRUE;
                FC_LogEvent(
                    eCode      := E_EventCode.CRIT_INV_CHECK_BELOW_THRESHOLD,
                    bRaised    := TRUE,
                    rParam1    := TO_REAL(fbCheckInv.uRespondedTotal),
                    rParam2    := TO_REAL(fbCheckInv.uConfiguredTotal),
                    uMachState := GVL_Main.MachineState
                );
                stState := E_StartupStatus.stError;
            END_IF
            // BUSY: fbCheckInv ainda varrendo — permanece no estado

    	// ────────────────────────────────────────────────────────────
    	// ────────────────────────────────────────────────────────────
    	E_StartupStatus.stWait_K1:																// DEBOUNCE K1

    		cmdK01 := TRUE;
    		auxRed := TRUE;																		// Status: aguardando K1 com debounce
    		auxYellow := FALSE;
    		auxGreen := FALSE;

    		TonDebounceK1(IN := auxK1_in, PT := TimeDebounceK1);
    		TonK1Timeout (IN := TRUE, PT := TimeK1Timeout);

    		IF TonDebounceK1.Q THEN
    		  debouncedK1 := TRUE;
    		ELSE
    		  debouncedK1 := FALSE;
    		END_IF

    		IF debouncedK1 AND (auxK1_in=TRUE) THEN
    		  // Para o timeout (não é mais necessário)
    		  TonK1Timeout(IN := FALSE);
    		  stState := E_StartupStatus.stWait_K2;												// Somente avança se K1 está estabilizado
    		  debouncedK2 := FALSE;
    		  TonDebounceK1(IN := FALSE, PT := TimeDebounceK1); 								// (Opcional) reseta timer
    		  auxRed := FALSE;																	// Status: aguardando K1 com debounce
    		  auxYellow := TRUE;
    		  auxGreen := FALSE;
    		  FC_LogEvent(
    			eCode      := E_EventCode.INFO_K1_CONFIRMED,
    			bRaised    := TRUE,
    			rParam1    := 0.0,
    			rParam2    := 0.0,
    			uMachState := GVL_Main.MachineState
    		  );
    		ELSIF TonK1Timeout.Q THEN															   // Se estourou timeout antes de confirmar debounce, gera alarme + evento crítico (1x)
    			GVL_Alarm.CRIT_K1_TIMEOUT:=TonK1Timeout.Q;
    			FC_LogEvent(
    				eCode      := E_EventCode.CRIT_K1_TIMEOUT,
    				bRaised    := TRUE,
    				rParam1    := 0.0,
    				rParam2    := 0.0,
    				uMachState := GVL_Main.MachineState
    			);
    		 	TonK1Timeout(IN := FALSE);
    			stState := E_StartupStatus.stError;
    		END_IF

    	// ────────────────────────────────────────────────────────────
    	// ────────────────────────────────────────────────────────────
    	E_StartupStatus.stWait_K2:

      		TonDebounceK2(IN := auxK2_in, PT := TimeDebounceK2);  								// debounce para K2_in
    		TonK2Timeout (IN := TRUE, PT := TimeK2Timeout);

    		IF TonDebounceK2.Q THEN																// tDebounce.Q será TRUE se K2_in estável
    		  debouncedK2 := TRUE;
    		ELSE
    		  debouncedK2 := FALSE;																// se K2_in voltar a false, reseta timer
    		END_IF

    		IF debouncedK2 AND (auxK2_in=TRUE) THEN
    		  TonK2Timeout(IN := FALSE);
    		  stState := E_StartupStatus.stDone;												// K2_ok e estável, processo de startup completo
    		  TonDebounceK2(IN := FALSE, PT := TimeDebounceK2); 								// (Opcional) reseta timer
    		  auxRed := FALSE;
    		  auxYellow := FALSE;
    		  auxGreen := TRUE;
    		  FC_LogEvent(
    			eCode      := E_EventCode.INFO_K2_CONFIRMED,
    			bRaised    := TRUE,
    			rParam1    := 0.0,
    			rParam2    := 0.0,
    			uMachState := GVL_Main.MachineState
    		  );
    		ELSIF TonK2Timeout.Q THEN 							// Se estourou timeout antes de confirmar debounce, gera alarme + evento crítico (1x)
    			GVL_Alarm.CRIT_K2_TIMEOUT:=TonK2Timeout.Q;
    			FC_LogEvent(
    				eCode      := E_EventCode.CRIT_K2_TIMEOUT,
    				bRaised    := TRUE,
    				rParam1    := 0.0,
    				rParam2    := 0.0,
    				uMachState := GVL_Main.MachineState
    			);
    		 	TonK2Timeout(IN := FALSE);
    			stState := E_StartupStatus.stError;
    		END_IF

    	// ────────────────────────────────────────────────────────────
    	// ────────────────────────────────────────────────────────────
    	E_StartupStatus.stDone:

    		stState := E_StartupStatus.stDone;
    		auxRed := FALSE;
    		auxYellow := FALSE;
    		auxGreen := TRUE;
    		FC_LogEvent(
    			eCode      := E_EventCode.INFO_STARTUP_DONE,
    			bRaised    := TRUE,
    			rParam1    := 0.0,
    			rParam2    := 0.0,
    			uMachState := GVL_Main.MachineState
    		);

    	// ────────────────────────────────────────────────────────────
    	// ────────────────────────────────────────────────────────────
    	E_StartupStatus.stError:
    		auxRed    := TRUE;
    		auxYellow := FALSE;
    		auxGreen  := FALSE;
    		// sai do case e no MainProgam vai para o estado ERRO

    END_CASE;

    //   Aplicar comandos calculados às saídas físicas / públicas
    GVL_Main.K1_out 		:= cmdK01;
    GVL_Main.LedRedOut 		:= auxRed;
    GVL_Main.LedYellowOut 	:= auxYellow;
    GVL_Main.LedGreenOut 	:= auxGreen;
END_FUNCTION_BLOCK

(* ---- FB_TurnOff.st ---- *)
(*
  FB_TurnOff - OPÇÃO B + MODO 1
  - FB NÃO usa GVL.
  - FB NÃO escreve setpoints, NÃO reseta PI, NÃO chama FB_WriteCom.
  - FB SÓ pede ações (pulsos) e decide transições.
  - Main executa: zerar setpoints + reset PI + chamadas FB_WriteCom.
*)
FUNCTION_BLOCK FB_TurnOff
VAR_INPUT
    xEnable          : BOOL;
    xStartResetEdge  : BOOL;

    xK2_in           : BOOL;

    rPt_kW           : REAL;
    xMeasDataOK      : BOOL;

    rP_Threshold_kW  : REAL := 0.5;
    tVerifyTimeout   : TIME := T#30S;
    tK2Timeout       : TIME := T#2S;
    uMaxWriteRetries : UINT := 3;

    // feedback das escritas (Main fornece)
    xCom1Done        : BOOL;
    xCom1Critical    : BOOL;
    xCom2Done        : BOOL;
    xCom2Critical    : BOOL;
END_VAR

VAR_OUTPUT
    // saídas físicas
    xK1_out          : BOOL;
    xK2_out          : BOOL;
    xLedRed          : BOOL;
    xLedYellow       : BOOL;
    xLedGreen        : BOOL;

    // pedidos ao Main (OPÇÃO B)
    xReqZeroSetpoints : BOOL;   // pulso 1 scan
    xReqResetPI       : BOOL;   // pulso 1 scan
    xReqResetCOM      : BOOL;   // pulso 1 scan
    xWriteZeroEnable  : BOOL;   // nível enquanto precisa escrever zero

    // transições
    xRequestStop     : BOOL;
    xRequestStart    : BOOL;

    // log 1 por transição
    xLogEvent        : BOOL;
    eLogCode         : E_EventCode;
    rLogParam1       : REAL;
    rLogParam2       : REAL;
END_VAR

VAR
    status              : E_TurnOffState := E_TurnOffState.TO_INIT;
    stPrevLogged     : E_TurnOffState := E_TurnOffState.TO_INIT;

    uRetry           : UINT := 0;

    tonVerify        : TON;
    tonK2            : TON;

    bInitPulseDone   : BOOL := FALSE;
END_VAR

    // defaults
    xRequestStop := FALSE;
    xRequestStart := FALSE;

    xReqZeroSetpoints := FALSE;
    xReqResetPI := FALSE;
    xReqResetCOM := FALSE;
    xWriteZeroEnable := FALSE;

    xLogEvent := FALSE;
    eLogCode := E_EventCode.EVT_NONE;
    rLogParam1 := 0.0;
    rLogParam2 := 0.0;

    IF NOT xEnable THEN
        status:= E_TurnOffState.TO_INIT;
        stPrevLogged := E_TurnOffState.TO_INIT;
        uRetry := 0;
        tonVerify(IN := FALSE);
        tonK2(IN := FALSE);
        bInitPulseDone := FALSE;

        xK1_out := FALSE;
        xK2_out := FALSE;
        xLedRed := FALSE;
        xLedYellow := FALSE;
        xLedGreen := FALSE;
        RETURN;
    END_IF

    // 1 log por transição (somente quando muda st)
    IF status<> stPrevLogged THEN
        stPrevLogged := status;
        xLogEvent := TRUE;
        CASE status OF
            E_TurnOffState.TO_INIT:        eLogCode := E_EventCode.INFO_TURNOFF_ENTRY;
            E_TurnOffState.TO_VERIFY:      eLogCode := E_EventCode.INFO_TURNOFF_ZERO_SENT;
            E_TurnOffState.TO_DISCONNECT:  eLogCode := E_EventCode.INFO_TURNOFF_EXPORT_CONFIRMED;
            E_TurnOffState.TO_CONFIRM:     eLogCode := E_EventCode.INFO_TURNOFF_K2_TRIPPED;
            E_TurnOffState.TO_DONE:        eLogCode := E_EventCode.INFO_TURNOFF_DONE;
        END_CASE
    END_IF

    CASE status OF

        E_TurnOffState.TO_INIT:
            xLedYellow := TRUE;  xLedGreen := FALSE; xLedRed := FALSE;
            xK1_out := TRUE;
            xK2_out := FALSE;

            tonVerify(IN := FALSE);
            tonK2(IN := FALSE);
            uRetry := 0;

            // pede ações UMA VEZ na entrada do TURNOFF (pulso)
            IF NOT bInitPulseDone THEN
                xReqZeroSetpoints := TRUE;
                xReqResetPI := TRUE;
                xReqResetCOM := TRUE;
                bInitPulseDone := TRUE;
            END_IF

            status:= E_TurnOffState.TO_WRITE_ZERO;

        E_TurnOffState.TO_WRITE_ZERO:
            xLedYellow := TRUE;  xLedGreen := FALSE; xLedRed := FALSE;
            xK1_out := TRUE;
            xK2_out := FALSE;

            // habilita escritas de zero no Main
            xWriteZeroEnable := TRUE;

            // aguarda resultado das duas COM (feedback do Main)
            IF xCom1Done AND xCom2Done THEN
                IF xCom1Critical OR xCom2Critical THEN
                    uRetry := uRetry + 1;

                    xLogEvent := TRUE;
                    eLogCode := E_EventCode.WARN_TURNOFF_WRITE_RETRY;
                    rLogParam1 := TO_REAL(uRetry);

                    IF uRetry >= uMaxWriteRetries THEN
                        xLogEvent := TRUE;
                        eLogCode := E_EventCode.CRIT_TURNOFF_WRITE_EXHAUSTED;
                        rLogParam1 := TO_REAL(uRetry);
                        xRequestStop := TRUE;
                    ELSE
                        // retry: pede reset COM + re-zero setpoints por segurança
                        xReqZeroSetpoints := TRUE;
                        xReqResetPI := TRUE;
                        xReqResetCOM := TRUE;
                        status:= E_TurnOffState.TO_WRITE_ZERO; // permanece, mas reinicia escrita no Main via ResetCOM
                    END_IF
                ELSE
                    status:= E_TurnOffState.TO_VERIFY;
                END_IF
            END_IF

        E_TurnOffState.TO_VERIFY:
            xLedYellow := TRUE;  xLedGreen := FALSE; xLedRed := FALSE;
            xK1_out := TRUE;
            xK2_out := FALSE;

            tonVerify(IN := TRUE, PT := tVerifyTimeout);

            IF xMeasDataOK AND (ABS(rPt_kW) < rP_Threshold_kW) THEN
                tonVerify(IN := FALSE);

                xLogEvent := TRUE;
                eLogCode := E_EventCode.INFO_TURNOFF_EXPORT_CONFIRMED;
                rLogParam1 := rPt_kW;
                rLogParam2 := rP_Threshold_kW;

                status:= E_TurnOffState.TO_DISCONNECT;
            END_IF

            IF tonVerify.Q THEN
                tonVerify(IN := FALSE);

                xLogEvent := TRUE;
                eLogCode := E_EventCode.CRIT_TURNOFF_VERIFY_TIMEOUT;
                rLogParam1 := rPt_kW;
                rLogParam2 := REAL#30.0;

                xRequestStop := TRUE;
            END_IF

        E_TurnOffState.TO_DISCONNECT:
            xLedYellow := TRUE;  xLedGreen := FALSE; xLedRed := FALSE;
            xK1_out := FALSE;
            xK2_out := TRUE;

            tonK2(IN := FALSE);
            status:= E_TurnOffState.TO_CONFIRM;

        E_TurnOffState.TO_CONFIRM:
            xLedYellow := TRUE;  xLedGreen := FALSE; xLedRed := FALSE;
            xK1_out := FALSE;
            xK2_out := TRUE;

            tonK2(IN := TRUE, PT := tK2Timeout);

            IF tonK2.Q THEN
                tonK2(IN := FALSE);

                IF xK2_in THEN
                    xLogEvent := TRUE;
                    eLogCode := E_EventCode.CRIT_TURNOFF_K2_NOT_OPENED;
                    xLedRed := TRUE;
                ELSE
                    xLogEvent := TRUE;
                    eLogCode := E_EventCode.INFO_TURNOFF_K2_CONFIRMED;
                END_IF

                status:= E_TurnOffState.TO_DONE;
            END_IF

        E_TurnOffState.TO_DONE:
            xK1_out := FALSE;
            xK2_out := TRUE;

            xLedGreen := FALSE;
            xLedYellow := TRUE;
            xLedRed := xK2_in;

            IF xStartResetEdge THEN
                xRequestStart := TRUE;

                // rearma interno p/ próxima vez
                status:= E_TurnOffState.TO_INIT;
                stPrevLogged := E_TurnOffState.TO_INIT;
                uRetry := 0;
                bInitPulseDone := FALSE;
            END_IF
    END_CASE
END_FUNCTION_BLOCK

(* ---- FB_ValidaDados.st ---- *)
(*═════════════════════════════════════════════════════════════════════
 FB_ValidaMedicao

 Valida medições do medidor trifásico via Modbus, aplica filtro
 passa-baixa e verifica consistência física das grandezas.

 ENTRADAS:
 - (nenhuma - lê de valorLido.WordArray via Modbus)

 SAÍDAS:
 - bDadosOK: TRUE se medições são válidas
 - bPoucosErros: TRUE se < 5 erros consecutivos
 - diagnosticCode: Código de falha (0 = OK)

 LÓGICA:
 1. Conversão de escalas (Modbus → unidades físicas)
 2. Validação de ranges individuais
 3. Validação cruzada (Pt vs soma, PF vs P/S)
 4. Detecção de congelamento
 5. Filtro passa-baixa exponencial (SOMENTE se validação OK)
 6. Atualização de variáveis globais (SOMENTE se validação OK)
 7. Janela de erros (5 consecutivos = FAIL_SAFE)
═════════════════════════════════════════════════════════════════════*)
FUNCTION_BLOCK FB_ValidaDados

VAR_INPUT
	Meas_Device     : E_MeasDeviceType;
END_VAR

VAR_OUTPUT
    bDadosOK		: BOOL 	:= FALSE;  // Dados aprovados
	bPoucosErros	: BOOL  := TRUE;  // IniciALARMente sem erros
END_VAR

VAR
	chint			: UN_chint;
	URP1439			: UN_URP1439;

	Ua    	    	: REAL := 0.0; // Volts
	Ub    	    	: REAL := 0.0; // Volts
	Uc    	    	: REAL := 0.0; // Volts

	Ia    	    	: REAL := 0.0; // amperes
	Ib    	    	: REAL := 0.0; // amperes
	Ic    	    	: REAL := 0.0; // amperes

	Pt    	    	: REAL := 0.0; // sem unidade
	Pa    	    	: REAL := 0.0; // sem unidade
	Pb    	    	: REAL := 0.0; // sem unidade
	Pc    	   		: REAL := 0.0; // sem unidade

	Qt    	    	: REAL := 0.0; // var
	Qa    	    	: REAL := 0.0; // var
	Qb    	    	: REAL := 0.0; // var
	Qc    	    	: REAL := 0.0; // var

	PFt    	    	: REAL := 0.0; // Watts
	PFa    	    	: REAL := 0.0; // Watts
	PFb    	    	: REAL := 0.0; // Watts
	PFc    	    	: REAL := 0.0; // Watts

	// Limites físicos (ajustar conforme instalação)
    PFMIN 			: REAL := 0.5;
    PFMAX 			: REAL := 1.0;

	// variaveis auxiliares
	Pt_last			: REAL;
	nErrors 		: UINT := 0;
	SomaP			: REAL;
	SomaQ 			: REAL;
	Calculado 		: REAL;
	Tolerancia  	: REAL :=0.05;
	Pt_lastatus		: REAL := 0.0;
    frozen_count 	: UINT := 0;
	FREEZE_THRESHOLD: UINT := 10;  		// 10 ciclos
	bFirstRun		: BOOL :=TRUE;
	Pt_filt 		: REAL :=0;
    Qt_filt 		: REAL :=0;
    PFt_filt 		: REAL :=0;

	// DETECÇÃO DE CONGELAMENTO
    tonFreeze       : TON;
    bFreezeAlarm    : BOOL := FALSE;
    bFreezePrev     : BOOL := FALSE;   // Para logar só na borda de subida
    FREEZE_TIME     : TIME := T#5S;
END_VAR

    // ═══════════════════════════════════════════════════════════════
    // 1. RESET DE ESTADO
    // ═══════════════════════════════════════════════════════════════

    GVL_Alarm.ALARM_MEAS_RANGE_ERROR := FALSE;

    // ═══════════════════════════════════════════════════════════════
    // 2. CONVERSÃO DE ESCALAS
    // ═══════════════════════════════════════════════════════════════

    CASE Meas_Device OF

    	E_MeasDeviceType.CHINT_DTSU666 :

    		Ua  := chint.EmReal.Ua * 0.1;			// em Volts
    		Ub  := chint.EmReal.Ub * 0.1;			// em Volts
    		Uc  := chint.EmReal.Uc * 0.1;			// em Volts

    		Ia  := chint.EmReal.Ia * 0.001;			// em Amperes
    		Ib  := chint.EmReal.Ib * 0.001;			// em Amperes
    		Ic  := chint.EmReal.Ic * 0.001;			// em Amperes

    		Pt  := chint.EmReal.Pt *0.0001;			// kW
    		Pa  := chint.EmReal.Pa *0.0001;			// kW
    		Pb  := chint.EmReal.Pb *0.0001;			// kW
    		Pc  := chint.EmReal.Pc *0.0001;			// kW

    		Qt  := chint.EmReal.Qt *0.0001;			// kvar
    		Qa  := chint.EmReal.Qa *0.0001;			// kvar
    		Qb  := chint.EmReal.Qb *0.0001;			// kvar
    		Qc  := chint.EmReal.Qc *0.0001;			// xkvar

    		PFt := chint.EmReal.PFt *0.001;
    		PFa := chint.EmReal.PFa *0.001;
    		PFb := chint.EmReal.PFb *0.001;
    		PFc := chint.EmReal.PFc *0.001;

    	E_MeasDeviceType.RELAY_URP1439TU :
    		(*
    		14 registros - 28 words
    		PFa    	    : REAL := 0.0; // 0099H - Valor positivo: 0…16384 × (1/16384) e Valor negativo: 49151…65535 = -((65535 - valor lido) / 16384)
    		PFb    	    : REAL := 0.0; // 009AH - Valor positivo: 0…16384 × (1/16384) e Valor negativo: 49151…65535 = -((65535 - valor lido) / 16384)
    		PFc    	    : REAL := 0.0; // 009BH - Valor positivo: 0…16384 × (1/16384) e Valor negativo: 49151…65535 = -((65535 - valor lido) / 16384)
    		Reserved01  : REAL;        // 009CH - sem informação
    		Reserved02  : REAL;        // 009DH - sem informação
    		Reserved03  : REAL;        // 009EH - sem informação
    		Reserved04  : REAL;        // 009FH - sem informação
    		Ia    	    : REAL := 0.0; // 00A0H - 12…25.600 × (1/256) A (multiplicar por RTC)
    		Ib    	    : REAL := 0.0; // 00A1H - 12…25.600 × (1/256) A (multiplicar por RTC)
    		Ic    	    : REAL := 0.0; // 00A2H - 12…25.600 × (1/256) A (multiplicar por RTC)
    		Reserved05  : REAL;        // 00A3H - sem informação
    		Ua    	    : REAL := 0.0; // 00A4H - 256…64.000 × (1/128) Vca (multiplicar por RTP)
    		Ub    	    : REAL := 0.0; // 00A5H - 256…64.000 × (1/128) Vca (multiplicar por RTP)
    		Uc    	    : REAL := 0.0; // 00A6H - 256…64.000 × (1/128) Vca (multiplicar por RTP)
    		*)

    		PFa := URP1439.EmReal.PFa;
    		PFb := URP1439.EmReal.PFb;
    		PFc := URP1439.EmReal.PFc;

    		Ua  := URP1439.EmReal.Ua;				// em Volts
    		Ub  := URP1439.EmReal.Ub;				// em Volts
    		Uc  := URP1439.EmReal.Uc;				// em Volts

    		Ia  := URP1439.EmReal.Ia;				// em Amperes
    		Ib  := URP1439.EmReal.Ib;				// em Amperes
    		Ic  := URP1439.EmReal.Ic;				// em Amperes

    	E_MeasDeviceType.RELAY_URP6000:
    		// a definir

    	E_MeasDeviceType.RELAY_REMP_GD:
    		// a definir

    END_CASE

    // ═══════════════════════════════════════════════════════════════
    // 3. VALIDAÇÃO DE RANGES (SEM RETURN)
    // ═══════════════════════════════════════════════════════════════
    // validação de tensões

    IF (Ua < GVL_Pers.VMIN) OR (Ua > GVL_Pers.VMAX) THEN
        GVL_Alarm.ALARM_MEAS_RANGE_ERROR := TRUE;
    	FC_LogEvent(eCode:=E_EventCode.ALARM_MEAS_VOLTAGE_A_RANGE,bRaised:=TRUE,rParam1:=Ua,rParam2:=0.0,uMachState:= GVL_Main.MachineState);
    END_IF
    IF (Ub < GVL_Pers.VMIN) OR (Ub > GVL_Pers.VMAX) THEN
        GVL_Alarm.ALARM_MEAS_RANGE_ERROR := TRUE;
    	FC_LogEvent(eCode:=E_EventCode.ALARM_MEAS_VOLTAGE_B_RANGE,bRaised:=TRUE,rParam1:=Ub,rParam2:=0.0,uMachState:= GVL_Main.MachineState);
    END_IF
    IF (Uc < GVL_Pers.VMIN) OR (Uc > GVL_Pers.VMAX) THEN
        GVL_Alarm.ALARM_MEAS_RANGE_ERROR := TRUE;
    	FC_LogEvent(eCode:=E_EventCode.ALARM_MEAS_VOLTAGE_C_RANGE,bRaised:=TRUE,rParam1:=Uc,rParam2:=0.0,uMachState:= GVL_Main.MachineState);
    END_IF

    // validação de correntes
    IF (ABS(Ia) > GVL_Pers.IMAX) THEN
        GVL_Alarm.ALARM_MEAS_RANGE_ERROR := TRUE;
    	FC_LogEvent(eCode:=E_EventCode.ALARM_MEAS_CURRENT_A_RANGE,bRaised:=TRUE,rParam1:=Ia,rParam2:=0.0,uMachState:= GVL_Main.MachineState);
    END_IF
    IF (ABS(Ib) > GVL_Pers.IMAX) THEN
        GVL_Alarm.ALARM_MEAS_RANGE_ERROR := TRUE;
    	FC_LogEvent(eCode:=E_EventCode.ALARM_MEAS_CURRENT_B_RANGE,bRaised:=TRUE,rParam1:=Ib,rParam2:=0.0,uMachState:= GVL_Main.MachineState);
    END_IF
    IF (ABS(Ic) > GVL_Pers.IMAX) THEN
        GVL_Alarm.ALARM_MEAS_RANGE_ERROR := TRUE;
    	FC_LogEvent(eCode:=E_EventCode.ALARM_MEAS_CURRENT_C_RANGE,bRaised:=TRUE,rParam1:=Ic,rParam2:=0.0,uMachState:= GVL_Main.MachineState);
    END_IF

    // validação do fator das potencias
    IF (ABS(PFa) < PFMIN) OR (ABS(PFa) >PFMAX)  THEN
        GVL_Alarm.ALARM_MEAS_RANGE_ERROR := TRUE;
    	FC_LogEvent(eCode:=E_EventCode.ALARM_MEAS_PFA_RANGE,bRaised:=TRUE,rParam1:=PFa,rParam2:=0.0,uMachState:= GVL_Main.MachineState);
    END_IF
    IF (ABS(PFb) < PFMIN) OR (ABS(PFb) >PFMAX)  THEN
        GVL_Alarm.ALARM_MEAS_RANGE_ERROR := TRUE;
    	FC_LogEvent(eCode:=E_EventCode.ALARM_MEAS_PFB_RANGE,bRaised:=TRUE,rParam1:=PFb,rParam2:=0.0,uMachState:= GVL_Main.MachineState);
    END_IF
    IF (ABS(PFc) < PFMIN) OR (ABS(PFc) >PFMAX)  THEN
        GVL_Alarm.ALARM_MEAS_RANGE_ERROR := TRUE;
    	FC_LogEvent(eCode:=E_EventCode.ALARM_MEAS_PFC_RANGE,bRaised:=TRUE,rParam1:=PFc,rParam2:=0.0,uMachState:= GVL_Main.MachineState);
    END_IF

    IF Meas_Device = E_MeasDeviceType.CHINT_DTSU666 THEN
    	// validação de potencias ativas
    	IF (ABS(Pt) > GVL_Pers.PMAX) THEN
    		GVL_Alarm.ALARM_MEAS_RANGE_ERROR := TRUE;
    		FC_LogEvent(eCode:=E_EventCode.ALARM_MEAS_PT_RANGE,bRaised:=TRUE,rParam1:=Pt,rParam2:=0.0,uMachState:= GVL_Main.MachineState);
    	END_IF
    	IF (ABS(Pa) > GVL_Pers.PMAX) THEN
    		GVL_Alarm.ALARM_MEAS_RANGE_ERROR := TRUE;
    		FC_LogEvent(eCode:=E_EventCode.ALARM_MEAS_PA_RANGE,bRaised:=TRUE,rParam1:=Pa,rParam2:=0.0,uMachState:= GVL_Main.MachineState);
    	END_IF
    	IF (ABS(Pb) > GVL_Pers.PMAX) THEN
    		GVL_Alarm.ALARM_MEAS_RANGE_ERROR := TRUE;
    		FC_LogEvent(eCode:=E_EventCode.ALARM_MEAS_PB_RANGE,bRaised:=TRUE,rParam1:=Pb,rParam2:=0.0,uMachState:= GVL_Main.MachineState);
    	END_IF
    	IF (ABS(Pc) > GVL_Pers.PMAX) THEN
    		GVL_Alarm.ALARM_MEAS_RANGE_ERROR := TRUE;
    		FC_LogEvent(eCode:=E_EventCode.ALARM_MEAS_PC_RANGE,bRaised:=TRUE,rParam1:=Pc,rParam2:=0.0,uMachState:= GVL_Main.MachineState);
    	END_IF

    	// validação de potencias reativas
    	IF (ABS(Qt) > GVL_Pers.QMAX) THEN
    		GVL_Alarm.ALARM_MEAS_RANGE_ERROR := TRUE;
    		FC_LogEvent(eCode:=E_EventCode.ALARM_MEAS_QT_RANGE,bRaised:=TRUE,rParam1:=Qt,rParam2:=0.0,uMachState:= GVL_Main.MachineState);
    	END_IF
    	IF (ABS(Qa) > GVL_Pers.QMAX) THEN
    		GVL_Alarm.ALARM_MEAS_RANGE_ERROR := TRUE;
    		FC_LogEvent(eCode:=E_EventCode.ALARM_MEAS_QA_RANGE,bRaised:=TRUE,rParam1:=Qa,rParam2:=0.0,uMachState:= GVL_Main.MachineState);
    	END_IF
    	IF (ABS(Qb) > GVL_Pers.QMAX) THEN
    		GVL_Alarm.ALARM_MEAS_RANGE_ERROR := TRUE;
    		FC_LogEvent(eCode:=E_EventCode.ALARM_MEAS_QB_RANGE,bRaised:=TRUE,rParam1:=Qb,rParam2:=0.0,uMachState:= GVL_Main.MachineState);
    	END_IF
    	IF (ABS(Qc) > GVL_Pers.QMAX) THEN
    		GVL_Alarm.ALARM_MEAS_RANGE_ERROR := TRUE;
    		FC_LogEvent(eCode:=E_EventCode.ALARM_MEAS_QC_RANGE,bRaised:=TRUE,rParam1:=Qc,rParam2:=0.0,uMachState:= GVL_Main.MachineState);
    	END_IF

    	// validação do fator das potencias
    	IF (ABS(PFt) < PFMIN) OR (ABS(PFt) >PFMAX)  THEN
    		GVL_Alarm.ALARM_MEAS_RANGE_ERROR := TRUE;
    		FC_LogEvent(eCode:=E_EventCode.ALARM_MEAS_PFT_RANGE,bRaised:=TRUE,rParam1:=PFt,rParam2:=0.0,uMachState:= GVL_Main.MachineState);
    	END_IF
    END_IF

    // ═══════════════════════════════════════════════════════════════
    // 4. VALIDAÇÃO CRUZADA (SÓ SE NÃO HOUVER ERRO AINDA)
    // ═══════════════════════════════════════════════════════════════

    IF NOT GVL_Alarm.ALARM_MEAS_RANGE_ERROR THEN
    	// Só valida se Pa significativo (ex: > 1 kW)
    	IF ABS(Pa) > 1.0 THEN
    		Calculado := Ua * Ia * PFa / 1000;
    		IF ABS(Pa - Calculado) > (ABS(Pa) * Tolerancia) THEN  // ✅ Usa Pa, não Calculado
    			GVL_Alarm.ALARM_MEAS_RANGE_ERROR := TRUE;
    			FC_LogEvent(eCode:=E_EventCode.ALARM_MEAS_PA_XCHECK_FAIL,bRaised:=TRUE,rParam1:=Pa,rParam2:=0.0,uMachState:= GVL_Main.MachineState);
    		END_IF
    	END_IF

    	// Repetir para Pb e Pc
    	IF ABS(Pb) > 1.0 THEN
    		Calculado := Ub * Ib * PFb / 1000;
    		IF ABS(Pb - Calculado) > (ABS(Pb) * Tolerancia) THEN
    			GVL_Alarm.ALARM_MEAS_RANGE_ERROR := TRUE;
    			FC_LogEvent(eCode:=E_EventCode.ALARM_MEAS_PB_XCHECK_FAIL,bRaised:=TRUE,rParam1:=Pb,rParam2:=0.0,uMachState:= GVL_Main.MachineState);
    		END_IF
    	END_IF

    	IF ABS(Pc) > 1.0 THEN
    		Calculado := Uc * Ic * PFc / 1000;
    		IF ABS(Pc - Calculado) > (ABS(Pc) * Tolerancia) THEN
    			GVL_Alarm.ALARM_MEAS_RANGE_ERROR := TRUE;
    			FC_LogEvent(eCode:=E_EventCode.ALARM_MEAS_PC_XCHECK_FAIL,bRaised:=TRUE,rParam1:=Pc,rParam2:=0.0,uMachState:= GVL_Main.MachineState);
    		END_IF
    	END_IF
    	// Pt = Pa + Pb + Pc
    	SomaP := Pa + Pb + Pc;
    	IF ABS(Pt) > 1.0 THEN  // ✅ Só valida se significativo
    		IF ABS(Pt - SomaP) > (ABS(Pt) * Tolerancia) THEN  // ✅ Usa Pt
    			GVL_Alarm.ALARM_MEAS_RANGE_ERROR := TRUE;
    			FC_LogEvent(eCode:=E_EventCode.ALARM_MEAS_PT_XCHECK_FAIL,bRaised:=TRUE,rParam1:=Pt,rParam2:=0.0,uMachState:= GVL_Main.MachineState);
    		END_IF
    	END_IF

    	// FPt com base nas potencias ativas e reativas
    	SomaQ:=Qa + Qb + Qc;
    	Calculado := SQRT((SomaP * SomaP)+ (SomaQ * SomaQ));
    	IF Calculado > 10 THEN 									// 1 kva
    		Calculado := SomaP / Calculado;
    		IF ABS(PFt - Calculado) > 0.05 THEN
    			GVL_Alarm.ALARM_MEAS_RANGE_ERROR := TRUE;
    			FC_LogEvent(eCode:=E_EventCode.ALARM_MEAS_PFT_XCHECK_FAIL,bRaised:=TRUE,rParam1:=PFt,rParam2:=0.0,uMachState:= GVL_Main.MachineState);
    		END_IF
    	END_IF
    END_IF;

    // ═══════════════════════════════════════════════════════════════
    // 5. DETECÇÃO DE CONGELAMENTO (OPCIONAL)
    // ═══════════════════════════════════════════════════════════════
    (*
    // Suspeita de congelamento — sem dependência de ALARM_MEAS_RANGE_ERROR
    bFrozenSuspect := (NOT bFirstRun)
                      AND (ABS(Pt - Pt_last) < 1.0);

    tonFreeze(IN := bFrozenSuspect, PT := FREEZE_TIME);

    bFreezeAlarm := tonFreeze.Q;

    // Loga SOMENTE na borda de subida — evita flood
    IF bFreezeAlarm AND NOT bFreezePrev THEN
        FC_LogEvent(
            eCode      := E_EventCode.ALARM_MEAS_FROZEN,
            bRaised    := TRUE,
            rParam1    := Pt,
            rParam2    := Pt_last,
            uMachState := GVL_Main.MachineState
        );
    END_IF

    // Loga recuperação na borda de descida
    IF NOT bFreezeAlarm AND bFreezePrev THEN
        FC_LogEvent(
            eCode      := E_EventCode.ALARM_MEAS_FROZEN,
            bRaised    := FALSE,
            rParam1    := Pt,
            rParam2    := Pt_last,
            uMachState := GVL_Main.MachineState
        );
    END_IF

    bFreezePrev  := bFreezeAlarm;
    Pt_last      := Pt;
    *)
    // ═══════════════════════════════════════════════════════════════
    // 6. TRATAMENTO FINAL DE ERRO/SUCESSO
    // ═══════════════════════════════════════════════════════==══════
    IF GVL_Alarm.ALARM_MEAS_RANGE_ERROR THEN

        nErrors := MIN(nErrors + 1, 5);	// Clamp em 5
        bDadosOK := FALSE;  // Dado atual é inválido

        IF nErrors < 5 THEN
            bPoucosErros := TRUE;    	// ⚠️ Ainda tolerável (1-4 erros)
        ELSE
            bPoucosErros := FALSE;   	// 🚨 Degradação crítica
        END_IF
        // ❌ NÃO atualiza variáveis globais (mantém último valor válido)
        // ❌ NÃO reseta filtro (preserva estado anterior)
    ELSE
    	// 1. Decrementa contador de erros (recuperação gradual)
        IF nErrors > 0 THEN
            nErrors := nErrors - 1;
        END_IF

        bDadosOK := TRUE;
        bPoucosErros := TRUE;

        // 2. FILTRO PASSA-BAIXA (Suavização de Medição)
        // ─────────────────────────────────────────────────────────
        IF bFirstRun THEN
            Pt_filt := Pt;
            Qt_filt := Qt;
            PFt_filt := PFt;
            bFirstRun := FALSE;
        ELSE
    		// Filtro exponencial: y[n] = α·x[n] + (1-α)·y[n-1]
            // ALPHA configurável (ex: 0.25 → ~3s para 95% do valor)
            Pt_filt := GVL_Pers.ALPHA * Pt + (1.0 - GVL_Pers.ALPHA) * Pt_filt;
            Qt_filt := GVL_Pers.ALPHA * Qt + (1.0 - GVL_Pers.ALPHA) * Qt_filt;
            PFt_filt := GVL_Pers.ALPHA * PFt + (1.0 - GVL_Pers.ALPHA) * PFt_filt;
        END_IF

    	// 3. ATUALIZAÇÃO DE VARIÁVEIS GLOBAIS
        // ──────────────────────────────────────────────────────────
    	GVL_Main.Ua  := Ua;				// em Volts
    	GVL_Main.Ub  := Ub;				// em Volts
    	GVL_Main.Uc  := Uc;				// em Volts

    	GVL_Main.Ia  := Ia;				// em Amperes
    	GVL_Main.Ib  := Ib;				// em Amperes
    	GVL_Main.Ic  := Ic;				// em Amperes

    	// Potência Ativa (FILTRADA para controle)
    	GVL_Main.Pt  := Pt_filt;			// kW
    	GVL_Main.Pa  := Pa;				// kW
    	GVL_Main.Pb  := Pb;				// kW
    	GVL_Main.Pc  := Pc;				// kW

    	// Potência Reativa (FILTRADA para controle de PF)
    	GVL_Main.Qt  := Qt_filt;			// kvar
    	GVL_Main.Qa  := Qa;				// kvar
    	GVL_Main.Qb  := Qb;				// kvar
    	GVL_Main.Qc  := Qc;				// kvar

        // Fator de Potência (FILTRADO para controle)
    	GVL_Main.PFt := PFt_filt;
    	GVL_Main.PFa := PFa;
    	GVL_Main.PFb := PFb;
    	GVL_Main.PFc := PFc;

    END_IF

END_FUNCTION_BLOCK

(* ---- FB_WriteCom.st ---- *)
(*
  FB_WriteCom
  ==========
  Objetivo
  --------
  Orquestrar a escrita Modbus em um conjunto de inversores de um mesmo canal de comunicação (ex.: COM1 ou COM2),
  garantindo escrita SEQUENCIAL e determinística, respeitando a limitação dos inversores Goodwe de aceitar apenas
  "um registro por vez".

  Conceito de "canais"
  --------------------
  No seu driver, cada canal de escrita (0..4) é disparado por um trigger dedicado:
      trigInv[invIndex, channelIndex]
  Ex.: channel 0 = Setpoint P, channel 1 = Setpoint PF, etc.
  A quantidade de canais a escrever é configurável por COM via nChannelsToWrite (1..5).

  Política de falha (definida)
  ----------------------------
  - Em ERRO/TIMEOUT NÃO-crítico: incrementa contadores e PULA o inversor (vai para o próximo),
    resetando ChIndex := 0 (não tenta escrever PF se P falhou).
  - Em ERRO/TIMEOUT crítico (contadores > máximos): sinaliza bCritical e encerra (Done=TRUE) para o MainProgram
    decidir transição para FAIL.

  Robustez
  --------
  - Este FB chama um FB_ModBus interno (1 transação por vez). Recomenda-se que o FB_ModBus implemente handshake
    com xBusy (TRIG -> WAIT_BUSY_ON -> WAIT_DONE) para evitar "Done fantasma".
  - Este FB NÃO faz FC_LogEvent/Alarm Manager diretamente por padrão: expõe dados (última falha, contadores)
    para o MainProgram aplicar a política de log sem spam.

  Reset / uso
  -----------
  - Use xEnable = TRUE apenas enquanto estiver no estado WRITE.
  - Ao sair de WRITE (xEnable=FALSE), o FB reseta e fica pronto para o próximo ciclo.
*)
FUNCTION_BLOCK FB_WriteCom
VAR_INPUT
    Reset			 : BOOL;
	tTimeout         : TIME := T#100MS;    // timeout por operação (por canal)
    nInverters       : UINT := 0;          // quantidade de inversores no COM (<=15)
    nChannelsToWrite : UINT := 2;          // 1..5 (canais 0..4)
    maxErrors        : UINT := 999;        // acima disso vira crítico
    maxTimeouts      : UINT := 999;        // acima disso vira crítico
END_VAR

VAR_IN_OUT
    trigInv    : ARRAY[1..15, 0..4] OF BOOL;                        // triggers por inversor e por canal (do MainProgram)
    pInvPtr    : ARRAY[1..15] OF POINTER TO ModbusSlaveComPort;     // ponteiros para os slaves (um por inversor)
END_VAR

VAR_OUTPUT
    Done        : BOOL;    // terminou varrer todos inversores (ou encerrou por crítico)
    bCritical   : BOOL;    // TRUE => MainProgram deve ir para FAIL
    ErrCount    : UINT;    // contagem acumulada de ERRO
    TmoCount    : UINT;    // contagem acumulada de TIMEOUT

    InvIndex    : UINT;    // índice atual (1..15) - diagnóstico
    ChIndex     : INT;     // canal atual (0..4)  - diagnóstico

    LastFailInv : UINT;            // último inversor que falhou (para log)
    LastFailCh  : INT;             // último canal que falhou (para log)
    FailRes 	: E_ModbusResult;  // ERRO ou TIMEOUT (para log)
END_VAR

VAR
    fbTx     : FB_ModBus;
END_VAR

    IF Reset THEN
    		// clamp defensivo
    		Done := FALSE;
    		bCritical := FALSE;
            InvIndex := 1;
            ChIndex := 0;
            ErrCount := 0;
            TmoCount := 0;
            LastFailInv := 0;
            LastFailCh := 0;
            FailRes := E_ModbusResult.BUSY;
    ELSE
            // terminou todos
            IF (InvIndex <= nInverters) THEN

    	        // Executa 1 canal por vez do inversor atual
                fbTx(
        	        tTimeout := tTimeout,
                    trigInv  := trigInv[InvIndex, ChIndex],
                    pSlave   := pInvPtr[InvIndex]^
                    );

                CASE fbTx.result OF
                    E_ModbusResult.DONE:
                        // avança canal dentro do inversor
                        IF ChIndex < (nChannelsToWrite - 1) THEN
                            ChIndex := ChIndex + 1;
                        ELSE
                            // terminou todos canais do inversor
                            ChIndex := 0;
                            InvIndex := InvIndex + 1;
                        END_IF

                    E_ModbusResult.ERRO:
                        ErrCount := ErrCount + 1;
                        LastFailInv := InvIndex;
                        LastFailCh := ChIndex;
                        FailRes := E_ModbusResult.ERRO;

                        IF ErrCount > maxErrors THEN
    							FailRes := E_ModbusResult.ERRO;
                                bCritical := TRUE;
    							Done := TRUE;
                            ELSE
                                // não-crítico: pula inversor inteiro
                                ChIndex := 0;
                                InvIndex := InvIndex + 1;
                            END_IF

                        E_ModbusResult.TIMEOUT:
                            TmoCount := TmoCount + 1;
                            LastFailInv := InvIndex;
                            LastFailCh := ChIndex;

                            IF TmoCount > maxTimeouts THEN
    							FailRes := E_ModbusResult.TIMEOUT;
                                bCritical := TRUE;
    							Done := TRUE;
                            ELSE
                                // não-crítico: pula inversor inteiro
                                ChIndex := 0;
                                InvIndex := InvIndex + 1;
                            END_IF
                    ELSE
                        // E_ModbusResult.BUSY = aguarda (não avança)
                    END_CASE
    		ELSE
    			Done := TRUE;
            END_IF
    END_IF
END_FUNCTION_BLOCK
